(* IEC 61131-3 sources: generating_plc_code_with_llms/Code#2/Bard/third run, 21 files *)

(* ---- 14.st ---- *)
// 7.6s
// 2
FUNCTION FC1001 :BOOL
VAR_INPUT
  MEW: REAL;
  SP: REAL;
  HYS: REAL;
END_VAR
VAR_IN_OUT
   OUT:BOOL;
END_VAR
VAR
   P_HYS: REAL;
END_VAR

FC1001 := TRUE;

IF MEW >= SP THEN
  P_HYS := SP * HYS;
  IF MEW - P_HYS > 0 THEN
    OUT := FALSE;
  ENDIF;
ELSE
  P_HYS := SP * HYS;
  IF MEW + P_HYS < 0 THEN
    OUT := TRUE;
  ENDIF;
ENDIF;

RETURN OUT;
END_FUNCTION

(* ---- 15.st ---- *)
// 9.77s
// 2
FUNCTION FC1002 :BOOL
VAR_INPUT
  E_A, SENSOR: BOOL;
  ZEITW: TIME;
END_VAR
VAR_IN_OUT
  ZEIT:TON;
  P_HU, P_AL: BOOL;
END_VAR

FC1002 := TRUE;

IF E_A THEN
  P1 := TRUE;
ELSE
  P1 := FALSE;
  ZEIT := 0;
  P_HU := FALSE;
  P_AL := FALSE;
ENDIF;

IF SENSOR THEN
  IF P1 THEN
    ZEIT := ZEIT + 1;
    IF ZEIT >= 3 THEN
      ZEIT := 0;
      WRITE("Warning signal switched off, alarm switched on");
      P_HU := FALSE;
      P_AL := TRUE;
    END_IF;
  ELSE
    WRITE("Ultrasonic sensor reports an approach");
    P_HU := TRUE;
  END_IF;
ELSE
  IF P_AL THEN
    WRITE("Alarm switched off, monitoring system switched off");
    P_AL := FALSE;
  END_IF;
END_IF;

RETURN FC1002;
END_FUNCTION

(* ---- 18.st ---- *)
// 8.20s
// 2
FUNCTION FC1003 : VOID
VAR_INPUT
  IN_R:REAL;
  IN_MAX, IN_MIN:REAL;
  OUT_MAX, OUT_MIN:REAL;
END_VAR
VAR_OUTPUT
  OUT_R:REAL;
  FEH:BOOL;
END_VAR
VAR_TEMP
  DIFF1, DIFF2:REAL;
END_VAR

FC1003:

DIFF1 := IN_MAX - IN_MIN;
DIFF2 := OUT_MAX - OUT_MIN;

IF (IN_R < IN_MIN OR IN_R > IN_MAX) THEN
  FEH := TRUE;
ELSE
  FEH := FALSE;
ENDIF;

IF FEH THEN
  OUT_R := 0.0;
ELSE
  OUT_R := (OUT_MIN + (IN_R - IN_MIN) / DIFF1 * DIFF2);
ENDIF;

RETURN;

END_FUNCTION

(* ---- 19.st ---- *)
// 9.97s
// 2
FUNCTION_BLOCK FB1005
VAR_INPUT
  START:BOOL;
  DICKE:REAL;
  V_MAX, V_MIN:REAL;
END_VAR
VAR_OUTPUT
  D_MAX, D_MIN:REAL;
  P1:BOOL;
END_VAR
VAR
  FO:BOOL;
END_VAR

FB1005:
VAR
  M_MAX: REAL;
  M_MIN: REAL;
END_VAR

M_MAX := 0;
M_MIN := 0;

IF START THEN
  M_MAX := M_MAX + DICK;
  IF M_MAX > V_MAX THEN
    P1 := TRUE;
  ENDIF;

  M_MIN := M_MIN + DICK;
  IF M_MIN < V_MIN THEN
    P1 := TRUE;
  ENDIF;

  FO := TRUE;
ELSE
  FO := FALSE;
ENDIF;

D_MAX := M_MAX;
D_MIN := M_MIN;

IF FO THEN
  FO := FALSE;
ELSE
  FO := TRUE;
ENDIF;

END_FUNCTION_BLOCK

(* ---- 20.st ---- *)
// 8.17s
// 2
FUNCTION_BLOCK INTERLOCK
  VAR_INPUT
    I1 : BOOL;
    I2 : BOOL;
    TL : TIME;
  END_VAR
  VAR_OUTPUT
    Q1 : BOOL;
    Q2 : BOOL;
  END_VAR
  VAR
    T1 : TOF;
    T2 : TOF;
  END_VAR

INTERLOCK:

IF I1 THEN
  T1 := TL;
  Q2 := FALSE;
ELSE
  Q1 := FALSE;
ENDIF;

IF I2 THEN
  T2 := TL;
  Q1 := FALSE;
ELSE
  Q2 := FALSE;
ENDIF;

IF T1.Q THEN
  Q1 := TRUE;
  T1 := 0;
ENDIF;

IF T2.Q THEN
  Q2 := TRUE;
  T2 := 0;
ENDIF;

END_FUNCTION_BLOCK

(* ---- 21.st ---- *)
// 25.93s
// 2
FUNCTION_BLOCK BURNER
VAR_INPUT
  IN : BOOL;
  STAGE2 : BOOL;
  OVER_TEMP : BOOL;
  OIL_TEMP : BOOL := TRUE;
  FLAME : BOOL;
  RST : BOOL;
  RST_TIMER : BOOL;
  PRE_HEAT_TIME : TIME := t#5s;
  PRE_VENT_TIME : TIME := t#15s;
  PRE_IGNITE_TIME : TIME := t#15s;
  POST_IGNITE_TIME : TIME := t#25s;
  STAGE2_DELAY : TIME := t#10s;
  SAFETY_TIME : TIME := t#5s;
  LOCKOUT_TIME : TIME := t#10s;
  MULTIPLE_IGNITION : BOOL := TRUE;
  KW1 : REAL;
  KW2 : REAL;
END_VAR
VAR_OUTPUT
  MOTOR : BOOL;
  COIL1 : BOOL;
  COIL2 : BOOL;
  PRE_HEAT : BOOL;
  IGNITE : BOOL;
  FAIL : BOOL;
  KWH : REAL;
  STATUS : BYTE;
END_VAR
VAR_IN_OUT
  RUNTIME1 : UDINT;
  RUNTIME2 : UDINT;
  CYCLES : UDINT;
END_VAR
VAR
  state : INT;
  last : TIME;
  tx : TIME;
  last_change : TIME;
  timer1 : TON;
  timer2 : TON;
  oil_temp_last : BOOL;
  cycles2 : UDINT;
END_VAR

BURNER:

IF OVER_TEMP THEN
  STATUS := 9;
  RETURN;
END_IF;

IF RST AND RST_TIMER THEN
  RST_TIMER := FALSE;
  state := 110;
  RETURN;
END_IF;

IF RST THEN
  RST_TIMER := TRUE;
  tx := LOCKOUT_TIME;
  RETURN;
END_IF;

IF IN AND NOT OVER_TEMP THEN
  state := 111;
ELSE
  IF state >= 111 THEN
    state := 110;
  END_IF;
  RETURN;
END_IF;

IF state = 110 THEN
  STATUS := 110;
  MOTOR := FALSE;
  COIL1 := FALSE;
  COIL2 := FALSE;
  PRE_HEAT := FALSE;
  IGNITE := FALSE;
  FAIL := FALSE;
  KWH := 0;
  RUNTIME1 := 0;
  RUNTIME2 := 0;
  CYCLES := 0;
ELSE
  IF state = 111 THEN
    STATUS := 111;
    PRE_HEAT := TRUE;
    timer1 := PRE_HEAT_TIME;
    tx := timer1;
    IF NOT OIL_TEMP AND (TIME_SINCE(last) > tx) THEN
      state := 110;
      FAIL := TRUE;
      STATUS := 1;
    END_IF;
    IF FLAME AND (TIME_SINCE(last) > tx) THEN
      state := 110;
      FAIL := TRUE;
      STATUS := 2;
    END_IF;
  ELSIF state = 112 THEN
    STATUS := 112;
    MOTOR := TRUE;
    COIL1 := TRUE;
    timer1 := PRE_VENT_TIME;
    tx := timer1;
    IF FLAME AND (TIME_SINCE(last) > tx) THEN
      state := 110;
      FAIL := TRUE;
      STATUS := 3;
    END_IF;
  ELSIF state = 113 THEN
    STATUS := 113;
    COIL2 := TRUE;
    IF NOT FLAME AND (TIME_SINCE(last) > SAFETY_TIME) THEN
      state := 110;
      FAIL := TRUE;
      STATUS := 4;
    END_IF;
    IF NOT FLAME AND MULTIPLE_IGNITION AND STAGE2 THEN
      IGNITE := TRUE;
      timer2 := PRE_IGNITE_TIME;
      tx := timer2;
    END_IF;
    IF STAGE2 AND (TIME_SINCE(last) > STAGE2_DELAY) THEN
      COIL2 := FALSE;
      cycles2 := cycles2 + 1;
      RUNTIME2 := RUNTIME2 + TIME_SPAN(last_change);
    last_change := TIME;
    IF STAGE2 THEN
      state := 112;
    ELSE
      state := 110;
    END_IF;
  ENDIF;
END_IF;

IF TIME_SINCE(last) > tx THEN
  IF state = 111 THEN
    MOTOR := TRUE;
    timer1 := PRE_VENT_TIME;
    tx := timer1;
    state := 112;
  ELSIF state = 112 THEN
    IGNITE := TRUE;
    timer2 := PRE_IGNITE_TIME;
    tx := timer2;
    state := 113;
  ELSIF state = 113 THEN
    IF MULTIPLE_IGNITION AND NOT FLAME THEN
      IGNITE := TRUE;
      timer2 := PRE_IGNITE_TIME;
      tx := timer2;
    ELSE
      KWH := KW1 + KW2 * cycles2;
      RUNTIME1 := RUNTIME1 + TIME_SPAN(last_change);
      CYCLES := CYCLES + cycles2;
      cycles2 := 0;
      state := 110;
    END_IF;
  END_IF;
END_IF;

timer1 := timer1 - TIME_SPAN(last);
timer2 := timer2 - TIME_SPAN(last);
last := TIME;

END_FUNCTION_BLOCK

(* ---- 1.st ---- *)
// 4.56s
// 2
VAR
  xAllOn : BOOL;
  xAllOff : BOOL;

  xAlarm1 : BOOL := FALSE;
  xAlarm2 : BOOL := FALSE;
END_VAR

PROGRAM main

VAR
  tmpSignal : BOOL;
END_VAR

IF xAllOn = TRUE THEN
  xAlarm1 := TRUE;
  xAlarm2 := TRUE;
  xAllOn := FALSE;
END_IF;

IF xAllOff = TRUE THEN
  xAlarm1 := FALSE;
  xAlarm2 := FALSE;
  xAllOff := FALSE;
END_IF;

END_PROGRAM

(* ---- 10.st ---- *)
// 5.38s
// 2
VAR_INPUT
  X : REAL;
END_VAR
VAR
  SigmoidValue : REAL;
END_VAR

PROGRAM main

SigmoidValue := 1.0 / (1.0 + exp(-X));

WRITE("Sigmoid value of " & REAL_TO_STRING(X) & ": " & REAL_TO_STRING(SigmoidValue));

END_PROGRAM

(* ---- 11.st ---- *)
// 6.01s
// 2
VAR_INPUT
  x : REAL;
END_VAR
VAR
  SignValue : REAL;
END_VAR

PROGRAM main

IF x > 0 THEN
  SignValue := 1.0;
ELSIF x < 0 THEN
  SignValue := -1.0;
ELSE
  SignValue := 0.0;
ENDIF;

WRITE("Sign of " & REAL_TO_STRING(x) & ": " & REAL_TO_STRING(SignValue));

END_PROGRAM

(* ---- 12.st ---- *)
// 5.71s
// 2
VAR
  X : REAL;
  HyperbolicSinValue : REAL;
END_VAR

PROGRAM main

HyperbolicSinValue := SIN(SQRT(2) * EXP(X));

WRITE("Hyperbolic sine value of " & REAL_TO_STRING(X) & ": " & REAL_TO_STRING(HyperbolicSinValue));

END_PROGRAM

(* ---- 13.st ---- *)
// 7.75s
// 2
VAR CONSTANT
  MAXNUMBERS : UINT := 99;
END_VAR

VAR
  aNumbers : ARRAY[0..MAXNUMBERS] OF INT;
  nCnt : INT := 0;
END_VAR

PROGRAM main

FOR i := 0 TO 99 DO
  aNumbers[i] := rnd(100);
END_FOR;

nCnt := 0;

REPEAT
  IF aNumbers[nCnt] = 10 THEN
    WRITE("The number 10 was found. Search aborted.");
    EXIT;
  ELSEIF nCnt = MAXNUMBERS THEN
    WRITE("The number " & INT_TO_STRING(searchNumber) & " was not found in the list.");
    EXIT;
  ENDIF;

  WRITE("Searching for the number " & INT_TO_STRING(searchNumber) & "...");
  WAIT;

  nCnt := nCnt + 1;
UNTIL (nCnt = MAXNUMBERS OR aNumbers[nCnt] = searchNumber) OR aNumbers[nCnt] = 10;

END_PROGRAM

(* ---- 16.st ---- *)
// 9.09s
// 2
VAR
  North_green : BOOL;
  North_yellow : BOOL;
  North_red : BOOL;
  East_green : BOOL;
  East_yellow : BOOL;
  East_red : BOOL;
  T1 : TON;
END_VAR

PROGRAM main

North_green := TRUE;
North_yellow := FALSE;
North_red := FALSE;
East_green := FALSE;
East_yellow := FALSE;
East_red := TRUE;

T1 := 5000;

WHILE TRUE DO
  WAIT ON T1;

  IF T1.Q THEN
    North_green := FALSE;
    North_yellow := TRUE;

    IF T1.CT >= 9500 THEN
      North_yellow := FALSE;
      North_red := TRUE;
      East_green := TRUE;
      East_yellow := FALSE;
    ELSE
      East_red := TRUE;
    ENDIF;
  ENDIF;
END_WHILE;

END_PROGRAM

(* ---- 17.st ---- *)
// 7.17s
// 2
VAR
  aiOutside : INT;
  aiHumidity: INT;
  sShowText : STRING[80];
END_VAR

PROGRAM weather_station

aiOutside := 23;
aiHumidity := 60;

IF (aiOutside < 18) THEN
  sShowText := "Cold";
ELSIF (aiOutside < 25) THEN
  IF (aiHumidity >= 40 AND aiHumidity <= 75) THEN
    sShowText := "Opt";
  ELSE
    sShowText := "Temp. OK";
  ENDIF;
ELSE
  sShowText := "Hot";
ENDIF;

WRITE(sShowText);

END_PROGRAM

(* ---- 2.st ---- *)
// 5.36s
// 2
VAR
N : INT := 5;
K : INT := 3;
i : INT := 0;
END_VAR

PROGRAM main
VAR
tmpResult : INT;
END_VAR

tmpResult := 1;

FOR i := 0 TO K - 1 DO
IF i > 0 THEN
tmpResult := tmpResult * (N - i);
END_IF;
END_FOR;

WRITE("The binomial coefficient for N = " & INT_TO_STRING(N) & " and K = " & INT_TO_STRING(K) & " is: " & INT_TO_STRING(tmpResult));

END_PROGRAM

(* ---- 3.st ---- *)
// 6.45s
// 2
VAR_INPUT
  X : INT;
END_VAR
VAR
  t1 : DINT;
  t2  : DINT;
  x_tmp : INT;
END_VAR

PROGRAM main
VAR
  result : INT;
END_VAR

IF X <= 1 THEN
  result := X;
ELSE
  t1 := 0;
  t2 := 1;

  FOR i := 2 TO X DO
    x_tmp := t1 + t2;
    t1 := t2;
    t2 := x_tmp;
  END_FOR;

  result := x_tmp;
END_IF;

WRITE("Fibonacci number for X = " & INT_TO_STRING(X) & " is: " & INT_TO_STRING(result));

END_PROGRAM

(* ---- 4.st ---- *)
// 6.8s
// 2
VAR
  aiLevel : INT;
  PercentLevel : UINT;
  doLow : BOOL := FALSE;
  doOk : BOOL := FALSE;
  doHigh : BOOL := FALSE;
  doAlarm : BOOL := FALSE;
END_VAR

PROGRAM main

CASE aiLevel
  WHEN 0 TO AI_LOW_LEVEL THEN
    doLow := TRUE;

  WHEN AI_LOW_LEVEL + 1 TO AI_OK_LEVEL THEN
    doLow := FALSE;
    doOk := TRUE;

  WHEN AI_OK_LEVEL + 1 TO AI_HIGH_LEVEL THEN
    doLow := FALSE;
    doOk := FALSE;
    doHigh := TRUE;

  WHEN AI_HIGH_LEVEL + 1 TO 32767 THEN
    doLow := FALSE;
    doOk := FALSE;
    doHigh := FALSE;
END_CASE;

IF PercentLevel < 1 THEN
  doAlarm := TRUE;
END_IF;

END_PROGRAM

(* ---- 5.st ---- *)
// 7.83s
// 2
VAR
  Start_Loop : BOOL := FALSE;
  one_hour : TIME := T#1h;
  One_Hour_Timer : TON;
  Gate_Open : BOOL := FALSE;
  Close_Gate_Inst : BOOL := FALSE;
  Sensed_Car : BOOL := FALSE;
  Sensed_Car_Inst : BOOL := FALSE;
  Sensed_App : BOOL := FALSE;
  Mobile_Inst : BOOL := FALSE;
  Auth : STRING := '';
  my_defined_str : STRING := 'abcd';
END_VAR

PROGRAM main

VAR
  tmpAuth : STRING;
END_VAR

One_Hour_Timer(PT := one_hour);

IF Start_Loop = FALSE THEN
  Start_Loop := TRUE;
  One_Hour_Timer.run;
END_IF;

IF One_Hour_Timer.Q AND Gate_Open = TRUE THEN
  Close_Gate_Inst := TRUE;
END_IF;

IF Sensed_Car = TRUE OR Sensed_App = TRUE THEN
  Sensed_Car_Inst := TRUE;
  tmpAuth := 'abcd';

  IF Auth = tmpAuth THEN
    Gate_Open := TRUE;
    CLOSE_GATE:;
  ELSE
    Gate_Open := FALSE;
  END_IF;
END_IF;

IF Mobile_Inst = TRUE THEN
  Sensed_App := TRUE;
  tmpAuth := 'abcd';

  IF Auth = tmpAuth THEN
    Gate_Open := TRUE;
    CLOSE_GATE:;
  ELSE
    Gate_Open := FALSE;
  END_IF;
END_IF;

END_PROGRAM

(* ---- 6.st ---- *)
// 9.74s
// 3
VAR
  CONSTANT
    WAIT : UINT := 0;
    TOP_POSITION : UINT := 1;
    BOTTOM_POSITION : UINT := 2;
    GETBOX : UINT := 3;
    UNLOAD_POSITION : UINT := 4;
    UNLOAD_BOX : UINT := 5;
  END_VAR

VAR
  (*-- digital outputs*)
  doConvTop: BOOL := FALSE;
  doConvBottom: BOOL := FALSE;
  doConvLift: BOOL := FALSE;
  doLiftTop: BOOL := FALSE;
  doLiftBottom: BOOL := FALSE;
  doLiftUnload: BOOL := FALSE;
  (*-- digital inputs*)
  diConvTop: BOOL;
  diConvBottom: BOOL;
  diLiftTop: BOOL;
  diLiftBottom: BOOL;
  diLiftUnload: BOOL;
  diBoxLift: BOOL;
  (*-- status variables*)
  selectLift: UINT := 0;
  ConvTopOn: BOOL := FALSE;
  ConvBottomOn: BOOL := FALSE;
END_VAR

PROGRAM main

IF diConvTop = TRUE THEN
  ConvTopOn := FALSE;
  doConvTop := FALSE;
  selectLift := BOTTOM_POSITION;
  doLiftBottom := TRUE;
  WAIT;
END_IF;

IF diConvBottom = TRUE THEN
  ConvBottomOn := FALSE;
  doConvBottom := FALSE;
  selectLift := TOP_POSITION;
  doLiftTop := TRUE;
  WAIT;
END_IF;

IF diLiftTop = TRUE AND selectLift = TOP_POSITION THEN
  doLiftTop := FALSE;
  doConvLift := TRUE;

  IF diBoxLift = TRUE THEN
    doConvLift := FALSE;
    selectLift := UNLOAD_POSITION;
    doLiftUnload := TRUE;
    WAIT;
  END_IF;
END_IF;

IF diLiftBottom = TRUE AND selectLift = BOTTOM_POSITION THEN
  doLiftBottom := FALSE;
  doConvLift := TRUE;

  IF diBoxLift = TRUE THEN
    doConvLift := FALSE;
    selectLift := UNLOAD_BOX;
    WAIT;
  END_IF;
END_IF;

IF diLiftUnload = TRUE AND selectLift = UNLOAD_POSITION THEN
  doLiftUnload := FALSE;
  doConvLift := FALSE;
  doConvBottom := TRUE;
  ConvBottomOn := TRUE;
  selectLift := 0;
  WAIT;
END_IF;

END_PROGRAM

(* ---- 7.st ---- *)
// 6.65s
// 2
VAR CONSTANT
  MAX_INDEX: USINT := 4;
END_VAR
VAR
  aWeights : ARRAY[0..MAX_INDEX] OF INT;
  iCnt : USINT;
  sumWeight : DINT := 0;
  avgWeight : INT;
END_VAR

PROGRAM main

FOR iCnt := 0 TO MAX_INDEX DO
  aWeights[iCnt] := 0;
  sumWeight := sumWeight + aWeights[iCnt];
END_FOR;

avgWeight := sumWeight / MAX_INDEX;

WRITE("Total Weight: " & INT_TO_STRING(sumWeight));
WRITE("Average Weight: " & INT_TO_STRING(avgWeight));

END_PROGRAM

(* ---- 8.st ---- *)
// 9.37s
// 2
VAR_INPUT
  X : REAL;
END_VAR
VAR
  w : REAL;
  i : INT;
  we : REAL;
  w1e : REAL;
  ewx : REAL;
  last : DWORD;
END_VAR

PROGRAM main

last := 1;
i := 0;
w := 1.0;
ewx := X;

WHILE last <> 0 DO
  we := 1.0 / ewx;
  w1e := w + we;
  ewx := X * w1e;
  last := abs(w - w1e);
  i := i + 1;
  IF i > 10 THEN
    WRITE("Error: Convergence not reached");
    STOP;
  END_IF;
END_WHILE;

WRITE("Lambert W of " & REAL_TO_STRING(X) & ": " & REAL_TO_STRING(w));

END_PROGRAM

(* ---- 9.st ---- *)
// 6.25s
// 2
VAR
  YEAR : INT;
  isLeapYear : BOOL;
END_VAR

PROGRAM main

isLeapYear := FALSE;

IF YEAR % 4 = 0 AND YEAR % 100 <> 0 THEN
  isLeapYear := TRUE;

ELSIF YEAR % 400 = 0 THEN
  isLeapYear := TRUE;
ENDIF;

WRITE("YEAR: " & INT_TO_STRING(YEAR) & " is a leap year?: " & BOOL_TO_STRING(isLeapYear));

END_PROGRAM
